// TIA Portal project "S7-1200_Conveyor_Sorting" (V17)

(* hardware
DEVICE "S7-1200 station_1"  S7-1200 Station
   slot 0: "Rack_0"  S7-1200 Rack  Rack  V1.0
   slot 1: "PLC_1"  CPU 1212C DC/DC/DC  6ES7 212-1AE40-0XB0  V4.2
DEVICE "HMI_1"  TP700 Comfort
   slot 0: "HMI_1"  TP700 Comfort  6AV2 124-0GC01-0AX0  17.0.0.0
   slot 1: "HMI_RT_1"  TP700 Comfort  6AV2 124-0GC01-0AX0  17.0.0.0
   slot 5: "HMI_1.IE_CP_1"  PROFINET Interface  17.0.0.0
      slot 1: "PROFINET Interface_1"  PROFINET Interface
         slot 1: "Port_1"  Port
         slot 2: "Port_2"  Port
   slot 7: "HMI_1.MPI/DP_CP_1"  MPI/DP Interface  17.0.0.0
*)

// ===== PLC "PLC_1"  CPU 1212C DC/DC/DC =====

VAR_GLOBAL   // PLC tag table "Default tag table"
   "StopPB" AT %I0.0 : Bool;
   "SensorEntry" AT %I0.1 : Bool;
   "SensorCheck" AT %I0.2 : Bool;
   "SensorSorter" AT %I0.3 : Bool;
   "FaultResetPB" AT %I0.4 : Bool;
   "FaultLamp" AT %Q0.0 : Bool;
   "EntryOccupiedLamp" AT %Q0.1 : Bool;
   "CheckOccupiedLamp" AT %Q0.2 : Bool;
   "SorterOccupiedLamp" AT %Q0.3 : Bool;
   "SortingActiveLamp" AT %Q0.4 : Bool;
   "Clock_Byte" AT %MB100 : Byte;
   "Clock_10Hz" AT %M100.0 : Bool;
   "Clock_5Hz" AT %M100.1 : Bool;
   "Clock_2.5Hz" AT %M100.2 : Bool;
   "Clock_2Hz" AT %M100.3 : Bool;
   "Clock_1.25Hz" AT %M100.4 : Bool;
   "Clock_1Hz" AT %M100.5 : Bool;
   "Clock_0.625Hz" AT %M100.6 : Bool;
   "Clock_0.5Hz" AT %M100.7 : Bool;
   "RemoveInvalidProduct" AT %M0.0 : Bool;
   "StartCommand" AT %M0.1 : Bool;
   "FaultResetHMI" AT %M0.2 : Bool;
END_VAR

DATA_BLOCK "Data_block_1"   // DB2
{ S7_Optimized_Access := 'TRUE' }
VERSION : 0.1
   VAR
      EntryOccupied : Bool;
      CheckOccupied : Bool;
      SorterOccupied : Bool;
      SortingActive : Bool;
      FaultActive : Bool;
      SystemRunning : Bool;
      EntryCheckTimeoutFault : Bool;
      CheckSorterTimeoutFault : Bool;
      LineStopped : Bool;
      CheckProductType : Int;
      SorterProductType : Int;
      ProductSelect : Int;
      ALine : Bool;
      BLine : Bool;
      RandomCounter : Int;
      RandomValue : Int;
      ProductACount : DInt;
      ProductBCount : DInt;
      InvalidProductFault : Bool;
      SensorCheckMemory : Bool;
      TotalProductsCount : DInt;
      AlarmWord : Word;
   END_VAR
BEGIN
END_DATA_BLOCK

// folder: System blocks/Program resources

DATA_BLOCK "IEC_Timer_0_DB_1"   // DB3
{ S7_Optimized_Access := 'TRUE' }
AUTHOR : Simatic
FAMILY : IEC
NAME : IEC_TMR
VERSION : 1.0
// stored: InstanceOfName IEC_TIMER
"IEC_TIMER"
BEGIN
END_DATA_BLOCK

DATA_BLOCK "IEC_Counter_0_DB"   // DB4
{ S7_Optimized_Access := 'TRUE' }
AUTHOR : Simatic
FAMILY : IEC
NAME : CNTR
VERSION : 1.0
// stored: InstanceOfName IEC_COUNTER
"IEC_COUNTER"
BEGIN
END_DATA_BLOCK

DATA_BLOCK "IEC_Timer_0_DB_3"   // DB5
{ S7_Optimized_Access := 'TRUE' }
AUTHOR : Simatic
FAMILY : IEC
NAME : IEC_TMR
VERSION : 1.0
// stored: InstanceOfName IEC_TIMER
"IEC_TIMER"
BEGIN
END_DATA_BLOCK

DATA_BLOCK "IEC_Timer_0_DB_4"   // DB6
{ S7_Optimized_Access := 'TRUE' }
AUTHOR : Simatic
FAMILY : IEC
NAME : IEC_TMR
VERSION : 1.0
// stored: InstanceOfName IEC_TIMER
"IEC_TIMER"
BEGIN
END_DATA_BLOCK

DATA_BLOCK "IEC_Counter_0_DB_1"   // DB7
{ S7_Optimized_Access := 'TRUE' }
AUTHOR : Simatic
FAMILY : IEC
NAME : CNTR
VERSION : 1.0
// stored: InstanceOfName IEC_COUNTER
"IEC_COUNTER"
BEGIN
END_DATA_BLOCK

DATA_BLOCK "IEC_Counter_0_DB_2"   // DB8
{ S7_Optimized_Access := 'TRUE' }
AUTHOR : Simatic
FAMILY : IEC
NAME : CNTR
VERSION : 1.0
// stored: InstanceOfName IEC_COUNTER
"IEC_COUNTER"
BEGIN
END_DATA_BLOCK

DATA_BLOCK "IEC_Timer_0_DB_2"   // DB9
{ S7_Optimized_Access := 'TRUE' }
AUTHOR : Simatic
FAMILY : IEC
NAME : IEC_TMR
VERSION : 1.0
// stored: InstanceOfName IEC_TIMER
"IEC_TIMER"
BEGIN
END_DATA_BLOCK

DATA_BLOCK "IEC_Timer_0_DB_5"   // DB10
{ S7_Optimized_Access := 'TRUE' }
AUTHOR : Simatic
FAMILY : IEC
NAME : IEC_TMR
VERSION : 1.0
// stored: InstanceOfName IEC_TIMER
"IEC_TIMER"
BEGIN
END_DATA_BLOCK

// folder: (top level)

ORGANIZATION_BLOCK "Main"   // OB1, LAD, ProgramCycle
TITLE = "Main Program Sweep (Cycle)"
{ S7_Optimized_Access := 'TRUE' }
VERSION : 0.1
   VAR_INPUT
      Initial_Call : Bool;   // Initial call of this OB
      Remanence : Bool;   // =True, if remanent data are available
   END_VAR
   VAR_TEMP   // added for the SCL form of the ladder/FBD networks
      _w1 : Bool;
      _w2 : Bool;
   END_VAR
BEGIN

REGION Network 1: Product Type Randomizer
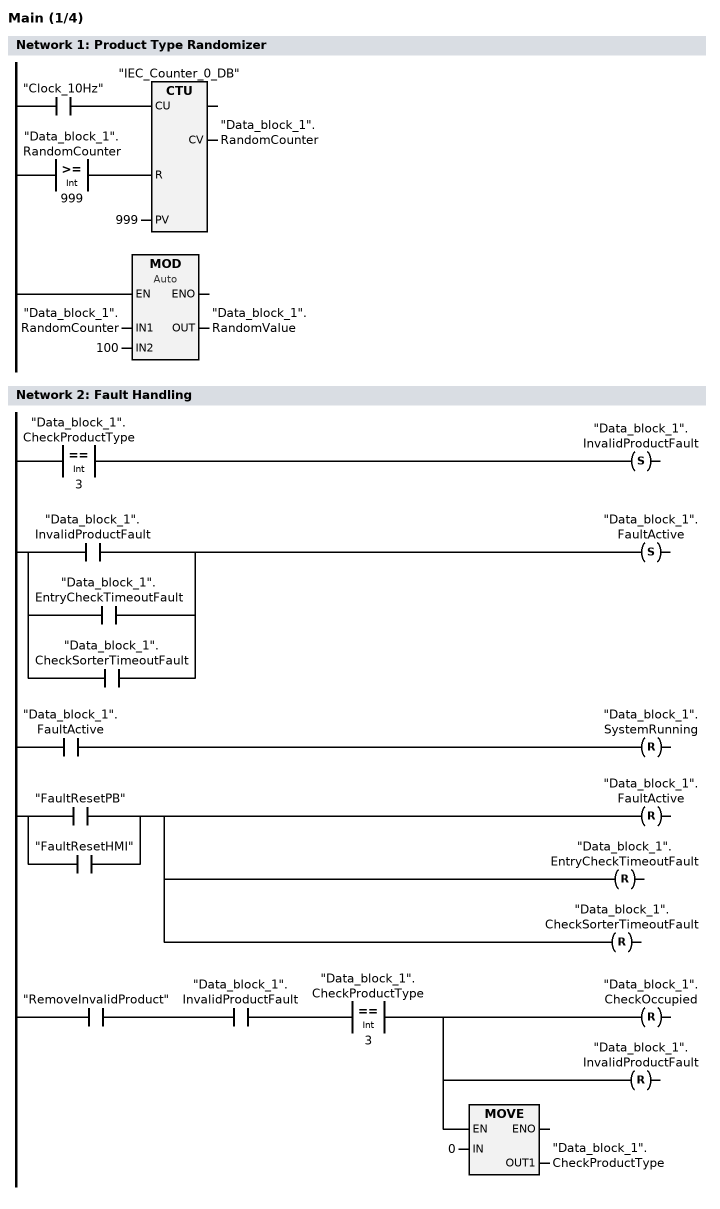
   "IEC_Counter_0_DB".CTU(CU := "Clock_10Hz",
                          R := "Data_block_1".RandomCounter >= 999,
                          PV := 999,
                          CV => "Data_block_1".RandomCounter);
   "Data_block_1".RandomValue := "Data_block_1".RandomCounter MOD 100;
END_REGION

REGION Network 2: Fault Handling
   RUNG wire#powerrail
      { S7_Templates := "SrcType := Int" } EQ_Contact(in1 := "Data_block_1".CheckProductType, in2 := 3)
      S_Coil( "Data_block_1".InvalidProductFault )
   END_RUNG
   RUNG wire#powerrail
      Contact( "Data_block_1".InvalidProductFault )
      wire#w1
      S_Coil( "Data_block_1".FaultActive )
   END_RUNG
   RUNG wire#powerrail
      Contact( "Data_block_1".EntryCheckTimeoutFault )
   END_RUNG wire#w1
   RUNG wire#powerrail
      Contact( "Data_block_1".CheckSorterTimeoutFault )
   END_RUNG wire#w1
   RUNG wire#powerrail
      Contact( "Data_block_1".FaultActive )
      R_Coil( "Data_block_1".SystemRunning )
   END_RUNG
   RUNG wire#powerrail
      Contact( "FaultResetPB" )
      wire#w2
      R_Coil( "Data_block_1".FaultActive )
   END_RUNG
   RUNG wire#powerrail
      Contact( "FaultResetHMI" )
   END_RUNG wire#w2
   RUNG wire#w2
      R_Coil( "Data_block_1".EntryCheckTimeoutFault )
   END_RUNG
   RUNG wire#w2
      R_Coil( "Data_block_1".CheckSorterTimeoutFault )
   END_RUNG
   RUNG wire#powerrail
      Contact( "RemoveInvalidProduct" )
      Contact( "Data_block_1".InvalidProductFault )
      { S7_Templates := "SrcType := Int" } EQ_Contact(in1 := "Data_block_1".CheckProductType, in2 := 3)
      wire#w3
      R_Coil( "Data_block_1".CheckOccupied )
   END_RUNG
   RUNG wire#w3
      R_Coil( "Data_block_1".InvalidProductFault )
   END_RUNG
   RUNG wire#w3
      Move(in := 0, out1 => "Data_block_1".CheckProductType)
   END_RUNG
   // the same network as SCL:
   IF "Data_block_1".CheckProductType = 3 THEN "Data_block_1".InvalidProductFault := TRUE; END_IF;
   IF "Data_block_1".InvalidProductFault OR "Data_block_1".EntryCheckTimeoutFault OR "Data_block_1".CheckSorterTimeoutFault THEN
       "Data_block_1".FaultActive := TRUE;
   END_IF;
   IF "Data_block_1".FaultActive THEN "Data_block_1".SystemRunning := FALSE; END_IF;
   IF "FaultResetPB" OR "FaultResetHMI" THEN
       "Data_block_1".FaultActive := FALSE;
       "Data_block_1".EntryCheckTimeoutFault := FALSE;
       "Data_block_1".CheckSorterTimeoutFault := FALSE;
   END_IF;
   IF "RemoveInvalidProduct" AND "Data_block_1".InvalidProductFault AND ("Data_block_1".CheckProductType = 3) THEN
       "Data_block_1".CheckOccupied := FALSE;
   END_IF;
   #_w1 := "RemoveInvalidProduct" AND "Data_block_1".InvalidProductFault AND ("Data_block_1".CheckProductType = 3);
   IF #_w1 THEN
       "Data_block_1".InvalidProductFault := FALSE;
       "Data_block_1".CheckProductType := 0;
   END_IF;
END_REGION

REGION Network 3: Alarm Word Mapping
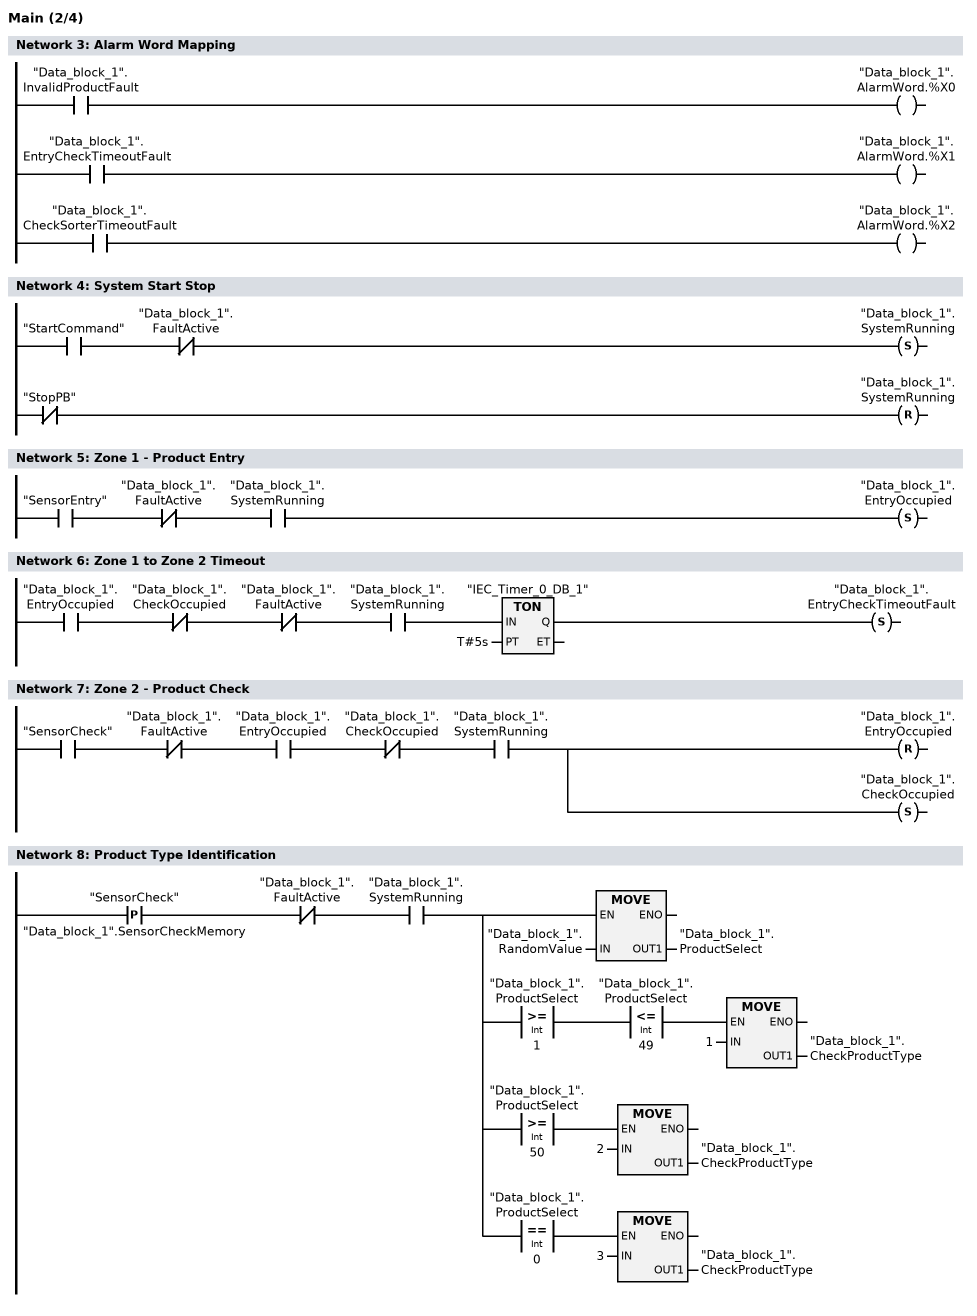
   RUNG wire#powerrail
      Contact( "Data_block_1".InvalidProductFault )
      Coil( "Data_block_1".AlarmWord.%X0 )
   END_RUNG
   RUNG wire#powerrail
      Contact( "Data_block_1".EntryCheckTimeoutFault )
      Coil( "Data_block_1".AlarmWord.%X1 )
   END_RUNG
   RUNG wire#powerrail
      Contact( "Data_block_1".CheckSorterTimeoutFault )
      Coil( "Data_block_1".AlarmWord.%X2 )
   END_RUNG
   // the same network as SCL:
   "Data_block_1".AlarmWord.%X0 := "Data_block_1".InvalidProductFault;
   "Data_block_1".AlarmWord.%X1 := "Data_block_1".EntryCheckTimeoutFault;
   "Data_block_1".AlarmWord.%X2 := "Data_block_1".CheckSorterTimeoutFault;
END_REGION

REGION Network 4: System Start Stop
   RUNG wire#powerrail
      Contact( "StartCommand" )
      I_Contact( "Data_block_1".FaultActive )
      S_Coil( "Data_block_1".SystemRunning )
   END_RUNG
   RUNG wire#powerrail
      I_Contact( "StopPB" )
      R_Coil( "Data_block_1".SystemRunning )
   END_RUNG
   // the same network as SCL:
   IF "StartCommand" AND NOT "Data_block_1".FaultActive THEN "Data_block_1".SystemRunning := TRUE; END_IF;
   IF NOT "StopPB" THEN "Data_block_1".SystemRunning := FALSE; END_IF;
END_REGION

REGION Network 5: Zone 1 - Product Entry
   RUNG wire#powerrail
      Contact( "SensorEntry" )
      I_Contact( "Data_block_1".FaultActive )
      Contact( "Data_block_1".SystemRunning )
      S_Coil( "Data_block_1".EntryOccupied )
   END_RUNG
   // the same network as SCL:
   IF "SensorEntry" AND NOT "Data_block_1".FaultActive AND "Data_block_1".SystemRunning THEN
       "Data_block_1".EntryOccupied := TRUE;
   END_IF;
END_REGION

REGION Network 6: Zone 1 to Zone 2 Timeout
   "IEC_Timer_0_DB_1".TON(IN := "Data_block_1".EntryOccupied AND NOT "Data_block_1".CheckOccupied AND NOT "Data_block_1".FaultActive AND "Data_block_1".SystemRunning,
                          PT := T#5s);
   IF "IEC_Timer_0_DB_1".Q THEN "Data_block_1".EntryCheckTimeoutFault := TRUE; END_IF;
END_REGION

REGION Network 7: Zone 2 - Product Check
   RUNG wire#powerrail
      Contact( "SensorCheck" )
      I_Contact( "Data_block_1".FaultActive )
      Contact( "Data_block_1".EntryOccupied )
      I_Contact( "Data_block_1".CheckOccupied )
      Contact( "Data_block_1".SystemRunning )
      wire#w1
      R_Coil( "Data_block_1".EntryOccupied )
   END_RUNG
   RUNG wire#w1
      S_Coil( "Data_block_1".CheckOccupied )
   END_RUNG
   // the same network as SCL:
   #_w1 := "SensorCheck" AND NOT "Data_block_1".FaultActive AND "Data_block_1".EntryOccupied AND NOT "Data_block_1".CheckOccupied AND "Data_block_1".SystemRunning;
   IF #_w1 THEN
       "Data_block_1".EntryOccupied := FALSE;
       "Data_block_1".CheckOccupied := TRUE;
   END_IF;
END_REGION

REGION Network 8: Product Type Identification
   RUNG wire#powerrail
      P_Contact(operand := "SensorCheck", bit := "Data_block_1".SensorCheckMemory)
      I_Contact( "Data_block_1".FaultActive )
      Contact( "Data_block_1".SystemRunning )
      wire#w1
      Move(in := "Data_block_1".RandomValue, out1 => "Data_block_1".ProductSelect)
   END_RUNG
   RUNG wire#w1
      { S7_Templates := "SrcType := Int" } GE_Contact(in1 := "Data_block_1".ProductSelect, in2 := 1)
      { S7_Templates := "SrcType := Int" } LE_Contact(in1 := "Data_block_1".ProductSelect, in2 := 49)
      Move(in := 1, out1 => "Data_block_1".CheckProductType)
   END_RUNG
   RUNG wire#w1
      { S7_Templates := "SrcType := Int" } GE_Contact(in1 := "Data_block_1".ProductSelect, in2 := 50)
      Move(in := 2, out1 => "Data_block_1".CheckProductType)
   END_RUNG
   RUNG wire#w1
      { S7_Templates := "SrcType := Int" } EQ_Contact(in1 := "Data_block_1".ProductSelect, in2 := 0)
      Move(in := 3, out1 => "Data_block_1".CheckProductType)
   END_RUNG
   // the same network as SCL:
   #_w1 := "SensorCheck" AND NOT "Data_block_1".SensorCheckMemory;   // rising edge of "SensorCheck"
   "Data_block_1".SensorCheckMemory := "SensorCheck";
   #_w2 := #_w1 AND NOT "Data_block_1".FaultActive AND "Data_block_1".SystemRunning;
   IF #_w2 THEN "Data_block_1".ProductSelect := "Data_block_1".RandomValue; END_IF;
   IF #_w2 AND ("Data_block_1".ProductSelect >= 1) AND ("Data_block_1".ProductSelect <= 49) THEN
       "Data_block_1".CheckProductType := 1;
   END_IF;
   IF #_w2 AND ("Data_block_1".ProductSelect >= 50) THEN "Data_block_1".CheckProductType := 2; END_IF;
   IF #_w2 AND ("Data_block_1".ProductSelect = 0) THEN "Data_block_1".CheckProductType := 3; END_IF;
END_REGION

REGION Network 9: Zone 2 to Zone 3 Timeout
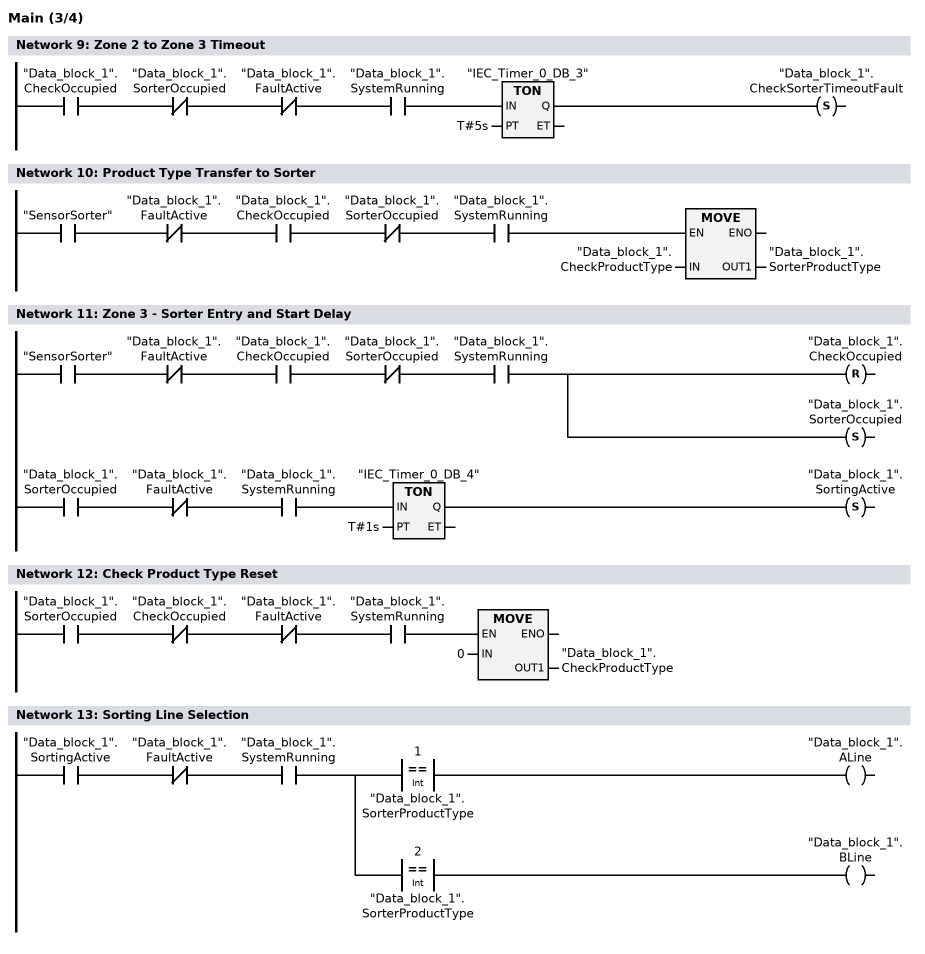
   "IEC_Timer_0_DB_3".TON(IN := "Data_block_1".CheckOccupied AND NOT "Data_block_1".SorterOccupied AND NOT "Data_block_1".FaultActive AND "Data_block_1".SystemRunning,
                          PT := T#5s);
   IF "IEC_Timer_0_DB_3".Q THEN "Data_block_1".CheckSorterTimeoutFault := TRUE; END_IF;
END_REGION

REGION Network 10: Product Type Transfer to Sorter
   RUNG wire#powerrail
      Contact( "SensorSorter" )
      I_Contact( "Data_block_1".FaultActive )
      Contact( "Data_block_1".CheckOccupied )
      I_Contact( "Data_block_1".SorterOccupied )
      Contact( "Data_block_1".SystemRunning )
      Move(in := "Data_block_1".CheckProductType, out1 => "Data_block_1".SorterProductType)
   END_RUNG
   // the same network as SCL:
   IF "SensorSorter" AND NOT "Data_block_1".FaultActive AND "Data_block_1".CheckOccupied AND NOT "Data_block_1".SorterOccupied AND "Data_block_1".SystemRunning THEN
       "Data_block_1".SorterProductType := "Data_block_1".CheckProductType;
   END_IF;
END_REGION

REGION Network 11: Zone 3 - Sorter Entry and Start Delay
   #_w1 := "SensorSorter" AND NOT "Data_block_1".FaultActive AND "Data_block_1".CheckOccupied AND NOT "Data_block_1".SorterOccupied AND "Data_block_1".SystemRunning;
   IF #_w1 THEN
       "Data_block_1".CheckOccupied := FALSE;
       "Data_block_1".SorterOccupied := TRUE;
   END_IF;
   "IEC_Timer_0_DB_4".TON(IN := "Data_block_1".SorterOccupied AND NOT "Data_block_1".FaultActive AND "Data_block_1".SystemRunning,
                          PT := T#1s);
   IF "IEC_Timer_0_DB_4".Q THEN "Data_block_1".SortingActive := TRUE; END_IF;
END_REGION

REGION Network 12: Check Product Type Reset
   RUNG wire#powerrail
      Contact( "Data_block_1".SorterOccupied )
      I_Contact( "Data_block_1".CheckOccupied )
      I_Contact( "Data_block_1".FaultActive )
      Contact( "Data_block_1".SystemRunning )
      Move(in := 0, out1 => "Data_block_1".CheckProductType)
   END_RUNG
   // the same network as SCL:
   IF "Data_block_1".SorterOccupied AND NOT "Data_block_1".CheckOccupied AND NOT "Data_block_1".FaultActive AND "Data_block_1".SystemRunning THEN
       "Data_block_1".CheckProductType := 0;
   END_IF;
END_REGION

REGION Network 13: Sorting Line Selection
   RUNG wire#powerrail
      Contact( "Data_block_1".SortingActive )
      I_Contact( "Data_block_1".FaultActive )
      Contact( "Data_block_1".SystemRunning )
      wire#w1
      { S7_Templates := "SrcType := Int" } EQ_Contact(in1 := 1, in2 := "Data_block_1".SorterProductType)
      Coil( "Data_block_1".ALine )
   END_RUNG
   RUNG wire#w1
      { S7_Templates := "SrcType := Int" } EQ_Contact(in1 := 2, in2 := "Data_block_1".SorterProductType)
      Coil( "Data_block_1".BLine )
   END_RUNG
   // the same network as SCL:
   #_w1 := "Data_block_1".SortingActive AND NOT "Data_block_1".FaultActive AND "Data_block_1".SystemRunning;
   "Data_block_1".ALine := #_w1 AND (1 = "Data_block_1".SorterProductType);
   "Data_block_1".BLine := #_w1 AND (2 = "Data_block_1".SorterProductType);
END_REGION

REGION Network 14: Sorting Process and Counters
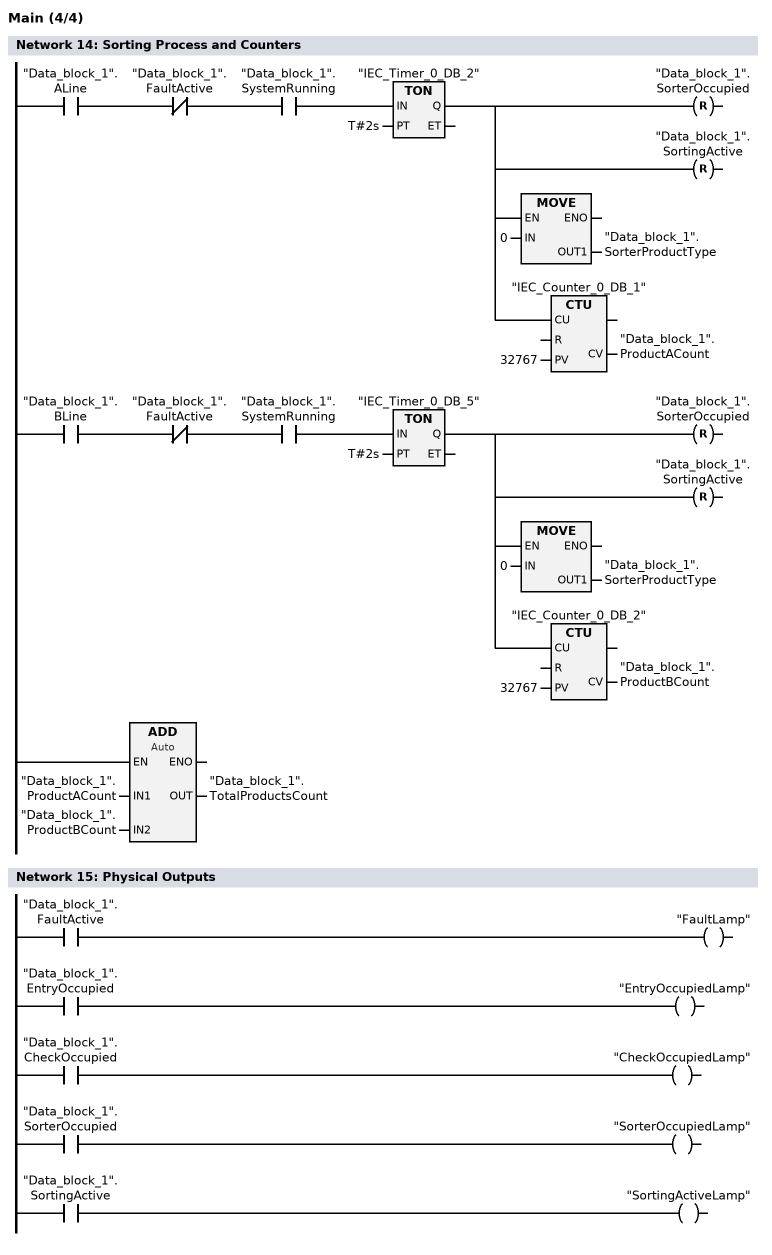
   "IEC_Timer_0_DB_2".TON(IN := "Data_block_1".ALine AND NOT "Data_block_1".FaultActive AND "Data_block_1".SystemRunning,
                          PT := T#2s);
   IF "IEC_Timer_0_DB_2".Q THEN
       "Data_block_1".SorterOccupied := FALSE;
       "Data_block_1".SortingActive := FALSE;
       "Data_block_1".SorterProductType := 0;
   END_IF;
   "IEC_Counter_0_DB_1".CTU(CU := "IEC_Timer_0_DB_2".Q, PV := 32767, CV => "Data_block_1".ProductACount);
   "IEC_Timer_0_DB_5".TON(IN := "Data_block_1".BLine AND NOT "Data_block_1".FaultActive AND "Data_block_1".SystemRunning,
                          PT := T#2s);
   IF "IEC_Timer_0_DB_5".Q THEN
       "Data_block_1".SorterOccupied := FALSE;
       "Data_block_1".SortingActive := FALSE;
       "Data_block_1".SorterProductType := 0;
   END_IF;
   "IEC_Counter_0_DB_2".CTU(CU := "IEC_Timer_0_DB_5".Q, PV := 32767, CV => "Data_block_1".ProductBCount);
   "Data_block_1".TotalProductsCount := "Data_block_1".ProductACount + "Data_block_1".ProductBCount;
END_REGION

REGION Network 15: Physical Outputs
   RUNG wire#powerrail
      Contact( "Data_block_1".FaultActive )
      Coil( "FaultLamp" )
   END_RUNG
   RUNG wire#powerrail
      Contact( "Data_block_1".EntryOccupied )
      Coil( "EntryOccupiedLamp" )
   END_RUNG
   RUNG wire#powerrail
      Contact( "Data_block_1".CheckOccupied )
      Coil( "CheckOccupiedLamp" )
   END_RUNG
   RUNG wire#powerrail
      Contact( "Data_block_1".SorterOccupied )
      Coil( "SorterOccupiedLamp" )
   END_RUNG
   RUNG wire#powerrail
      Contact( "Data_block_1".SortingActive )
      Coil( "SortingActiveLamp" )
   END_RUNG
   // the same network as SCL:
   "FaultLamp" := "Data_block_1".FaultActive;
   "EntryOccupiedLamp" := "Data_block_1".EntryOccupied;
   "CheckOccupiedLamp" := "Data_block_1".CheckOccupied;
   "SorterOccupiedLamp" := "Data_block_1".SorterOccupied;
   "SortingActiveLamp" := "Data_block_1".SortingActive;
END_REGION
END_ORGANIZATION_BLOCK

(* ===== HMI "HMI_RT_1" =====
system functions are stored by id; their names below are inferred from use
connection "HMI_Connection_2": ETHERNET, S7_1200_OMS

HMI tags "Default tag table"
   "Data_block_1_SystemRunning" : Bool = PLC Data_block_1.SystemRunning, 1 s
   "Data_block_1_FaultActive" : Bool = PLC Data_block_1.FaultActive, 1 s
   "CheckOccupiedLamp" : Bool = PLC CheckOccupiedLamp AT %Q0.2, 1 s
   "EntryOccupiedLamp" : Bool = PLC EntryOccupiedLamp AT %Q0.1, 1 s
   "SorterOccupiedLamp" : Bool = PLC SorterOccupiedLamp AT %Q0.3, 1 s
   "Data_block_1_CheckProductType" : Int = PLC Data_block_1.CheckProductType, 1 s
   "Data_block_1_SorterProductType" : Int = PLC Data_block_1.SorterProductType, 1 s
   "RemoveInvalidProduct" : Bool = PLC RemoveInvalidProduct AT %M0.0, 1 s
   "Data_block_1_ALine" : Bool = PLC Data_block_1.ALine, 1 s
   "Data_block_1_BLine" : Bool = PLC Data_block_1.BLine, 1 s
   "SensorCheck" : Bool = PLC SensorCheck AT %I0.2, 1 s
   "SensorSorter" : Bool = PLC SensorSorter AT %I0.3, 1 s
   "Data_block_1_TotalProductsCount" : DInt = PLC Data_block_1.TotalProductsCount, 1 s
   "Data_block_1_ProductACount" : DInt = PLC Data_block_1.ProductACount, 1 s
   "Data_block_1_ProductBCount" : DInt = PLC Data_block_1.ProductBCount, 1 s
   "Data_block_1_InvalidProductFault" : Bool = PLC Data_block_1.InvalidProductFault AT %DB1.DBX0.0, 1 s
   "Data_block_1_AlarmWord" : Word = PLC Data_block_1.AlarmWord, 1 s
   "FaultResetPB" : Bool = PLC FaultResetPB AT %I0.4, 1 s
   "FaultResetHMI" : Bool = PLC FaultResetHMI AT %M0.2, 1 s
   "StopPB" : Bool = PLC StopPB AT %I0.0, 1 s
   "SensorEntry" : Bool = PLC SensorEntry AT %I0.1, 1 s
   "FaultLamp" : Bool = PLC FaultLamp AT %Q0.0, 1 s
   "SortingActiveLamp" : Bool = PLC SortingActiveLamp AT %Q0.4, 1 s
   "Data_block_1_EntryOccupied" : Bool = PLC Data_block_1.EntryOccupied, 1 s
   "Data_block_1_CheckOccupied" : Bool = PLC Data_block_1.CheckOccupied, 1 s
   "Data_block_1_SorterOccupied" : Bool = PLC Data_block_1.SorterOccupied, 1 s
   "Data_block_1_SortingActive" : Bool = PLC Data_block_1.SortingActive, 1 s
   "Data_block_1_Zone1-Zone2Fault" : Bool = PLC Data_block_1.EntryCheckTimeoutFault, 1 s
   "Data_block_1_Zone2-Zone3Fault" : Bool = PLC Data_block_1.CheckSorterTimeoutFault, 1 s
   "StartCommand" : Bool = PLC StartCommand AT %M0.1, 1 s

discrete alarms
   1: 'Invalid product detected - remove product and reset fault', class Errors, trigger "Data_block_1_AlarmWord" bit 0
   2: 'Product timeout between ENTRY and CHECK', class Errors, trigger "Data_block_1_AlarmWord" bit 1
   3: 'Product timeout between CHECK and SORTER', class Errors, trigger "Data_block_1_AlarmWord" bit 2

graphic list "@DiagnosticsStates": 0 '@Diagnostics_StateGood'; 1 '@Diagnostics_StateBad'

Template "Template_1" 800x480
   Button "Exit" at 720,420 size 78x58; TextOff 'Exit'; PictureOff "ExitRuntime_TP700_Comfort_TR"; PictureOn "ExitRuntime_TP700_Comfort_TR"
      on Release: StopRuntime(0)
   Button "Template_Button_6" at 161,420 size 126x58; TextOff 'DIAGNOSTICS'
      on Click: ActivateScreen("Diagnostics", 0)
   Button "Template_Button_7" at 81,420 size 78x58; TextOff 'ALARMS'
      on Click: ActivateScreen("Alarms", 0)
   Button "Start screen" at 1,420 size 78x58; TextOff 'Start screen'; PictureOff "NavigateHome_TP700_Comfort_TR"; PictureOn "NavigateHome_TP700_Comfort_TR"
      on Click: ActivateScreen("Root screen", 0)

screen "Root screen" 800x480, template "Template_1"
   TextField "HmiScreenItemData" at 6,108 size 640x25; Text 'Text'
   TextField "Text field_1" at 218,1 size 402x34; Text 'CONVEYOR SORTING SYSTEM'
   TextField "Text field_2" at 13,40 size 84x23; Text 'SYSTEM:'
   TextField "Text field_3" at 90,40 size 89x23; Text 'STOPPED'
      Visibility <- "Data_block_1_SystemRunning"
      Appearance <- "Data_block_1_SystemRunning"
   TextField "Text field_4" at 90,40 size 91x23; Text 'RUNNING'
      Visibility <- "Data_block_1_SystemRunning"
      Appearance <- "Data_block_1_SystemRunning"
   Button "Button_1" at 47,76 size 96x32; TextOff 'START'
      on Press: SetBit("StartCommand")
      Visibility <- "Data_block_1_FaultActive"
      on Release: ResetBit("StartCommand")
   Button "Button_2" at 47,117 size 96x32; TextOff 'STOP'
      on Press: ResetBit("Data_block_1_SystemRunning")
      Visibility <- "Data_block_1_FaultActive"
   TextField "Text field_5" at 542,40 size 70x23; Text 'FAULT:'
   TextField "Text field_6" at 612,40 size 31x23; Text 'NO'
      Appearance <- "Data_block_1_FaultActive"
      Visibility <- "Data_block_1_FaultActive"
   TextField "Text field_7" at 604,40 size 73x23; Text 'ACTIVE'
      Appearance <- "Data_block_1_FaultActive"
      Visibility <- "Data_block_1_FaultActive"
   Circle "Circle_1" at 671,28 size 48x48
      Appearance <- "Data_block_1_FaultActive"
      Visibility <- "Data_block_1_FaultActive"
   Polygon "Polygon_2" at 572,298 size 21x14
      Appearance <- "Data_block_1_BLine"
   Polygon "Polygon_3" at 477,298 size 21x14
      Appearance <- "Data_block_1_ALine"
   TextField "Text field_8" at 555,312 size 65x23; Text 'B LINE'
   TextField "Text field_9" at 462,312 size 66x23; Text 'A LINE'
   Polygon "Polygon_4" at 320,199 size 13x20
      Appearance <- "SensorCheck"
   Polygon "Polygon_5" at 474,199 size 13x20
      Appearance <- "SensorSorter"
   TextField "Text field_10" at 186,199 size 93x23; Text 'PRODUCT'
   TextField "Text field_11" at 339,199 size 93x23; Text 'PRODUCT'
   TextField "Text field_12" at 492,199 size 93x23; Text 'PRODUCT'
   Circle "Circle_2" at 213,149 size 30x30
      Appearance <- "EntryOccupiedLamp"
   Circle "Circle_3" at 367,149 size 30x30
      Appearance <- "CheckOccupiedLamp"
   Circle "Circle_4" at 521,149 size 30x30
      Appearance <- "SorterOccupiedLamp"
   TextField "Text field_13" at 197,117 size 66x23; Text 'ENTRY'
   TextField "Text field_14" at 352,117 size 65x23; Text 'CHECK'
   TextField "Text field_15" at 498,117 size 78x23; Text 'SORTER'
   TextField "Text field_16" at 373,151 size 18x23; Text 'A'
      Visibility <- "Data_block_1_CheckProductType"
   TextField "Text field_17" at 528,151 size 18x23; Text 'A'
      Visibility <- "Data_block_1_SorterProductType"
   TextField "Text field_18" at 374,151 size 17x23; Text 'B'
      Visibility <- "Data_block_1_CheckProductType"
   TextField "Text field_19" at 529,151 size 17x23; Text 'B'
      Visibility <- "Data_block_1_SorterProductType"
   TextField "Text field_20" at 373,151 size 17x23; Text 'C'
      Visibility <- "Data_block_1_CheckProductType"
   TextField "Text field_21" at 29,280 size 78x23; Text 'TOTAL:'
   TextField "Text field_22" at 29,332 size 125x23; Text 'PRODUCT A:'
   TextField "Text field_23" at 29,374 size 124x23; Text 'PRODUCT B:'
   IOField "I/O field_1" at 97,276 size 96x32; FormatPattern 999999
      ProcessValue <- "Data_block_1_TotalProductsCount"
   IOField "I/O field_2" at 143,327 size 96x32; FormatPattern 999999
      ProcessValue <- "Data_block_1_ProductACount"
   IOField "I/O field_3" at 143,369 size 96x32; FormatPattern 999999
      ProcessValue <- "Data_block_1_ProductBCount"

screen "Alarms" 800x480, template "Template_1"
   TextField "Text field_1" at 260,9 size 266x23; Text 'ALARMS & FAULT HANDLING'
   AlarmView "Alarm view_1" at 23,98 size 761x241
   TextField "Text field_5" at 523,49 size 70x23; Text 'FAULT:'
   TextField "Text field_6" at 593,49 size 31x23; Text 'NO'
      Visibility <- "Data_block_1_FaultActive"
      Appearance <- "Data_block_1_FaultActive"
   TextField "Text field_7" at 585,49 size 73x23; Text 'ACTIVE'
      Visibility <- "Data_block_1_FaultActive"
      Appearance <- "Data_block_1_FaultActive"
   Circle "Circle_1" at 652,37 size 48x48
      Visibility <- "Data_block_1_FaultActive"
      Appearance <- "Data_block_1_FaultActive"
   TextField "Text field_2" at 98,49 size 84x23; Text 'SYSTEM:'
   TextField "Text field_3" at 175,49 size 89x23; Text 'STOPPED'
      Visibility <- "Data_block_1_SystemRunning"
      Appearance <- "Data_block_1_SystemRunning"
   TextField "Text field_4" at 175,49 size 91x23; Text 'RUNNING'
      Visibility <- "Data_block_1_SystemRunning"
      Appearance <- "Data_block_1_SystemRunning"
   Button "Button_1" at 151,379 size 96x32; TextOff 'RESET'
      on Press: SetBit("FaultResetHMI")
      on Release: ResetBit("FaultResetHMI")
      Visibility <- "Data_block_1_FaultActive"
   Button "Button_2" at 497,379 size 96x32; TextOff 'REMOVE'
      on Press: SetBit("RemoveInvalidProduct")
      on Release: ResetBit("RemoveInvalidProduct")
      Visibility <- "Data_block_1_InvalidProductFault"
   TextField "Text field_8" at 140,356 size 127x23; Text 'FAULT RESET'
      Visibility <- "Data_block_1_FaultActive"
   TextField "Text field_9" at 434,356 size 257x23; Text 'REMOVE INVALID PRODUCT'
      Visibility <- "Data_block_1_InvalidProductFault"

screen "Diagnostics" 800x480, template "Template_1"
   TextField "Text field_1" at 334,13 size 132x23; Text 'DIAGNOSTICS'
   TextField "Text field_2" at 40,51 size 157x23; Text 'DIGITAL INPUTS'
   TextField "Text field_3" at 38,84 size 76x23; Text 'Stop PB'
   TextField "Text field_4" at 38,111 size 120x23; Text 'Entry Sensor'
   TextField "Text field_5" at 38,138 size 126x23; Text 'Check Sensor'
   TextField "Text field_6" at 40,165 size 129x23; Text 'Sorter Sensor'
   TextField "Text field_7" at 40,191 size 109x23; Text 'Fault Reset'
   Circle "Circle_1" at 109,83 size 26x26
      Appearance <- "StopPB"
   Circle "Circle_2" at 147,108 size 26x26
      Appearance <- "SensorEntry"
   Circle "Circle_3" at 153,136 size 26x26
      Appearance <- "SensorCheck"
   Circle "Circle_4" at 157,164 size 26x26
      Appearance <- "SensorSorter"
   Circle "Circle_5" at 139,188 size 26x26
      Appearance <- "FaultResetPB"
   TextField "Text field_8" at 270,49 size 174x23; Text 'DIGITAL OUTPUTS'
   TextField "Text field_9" at 270,97 size 178x23; Text 'Entry Stage Yellow'
   TextField "Text field_10" at 270,120 size 177x23; Text 'Check Stage Green'
   TextField "Text field_11" at 270,143 size 179x23; Text 'Sorter Stage White'
   TextField "Text field_12" at 270,74 size 105x23; Text 'Fault Lamp'
   TextField "Text field_13" at 270,166 size 125x23; Text 'Sorting Lamp'
   Circle "Circle_6" at 365,72 size 26x26
      Appearance <- "FaultLamp"
   Circle "Circle_7" at 430,92 size 26x26
      Appearance <- "EntryOccupiedLamp"
   Circle "Circle_8" at 430,118 size 26x26
      Appearance <- "CheckOccupiedLamp"
   Circle "Circle_9" at 430,144 size 26x26
      Appearance <- "SorterOccupiedLamp"
   Circle "Circle_10" at 389,164 size 26x26
      Appearance <- "SortingActiveLamp"
   TextField "Text field_15" at 519,49 size 166x23; Text 'PROCESS STATUS'
   TextField "Text field_16" at 517,118 size 140x23; Text 'Entry Occupied'
   TextField "Text field_17" at 517,143 size 146x23; Text 'Check Occupied'
   TextField "Text field_18" at 517,166 size 149x23; Text 'Sorter Occupied'
   TextField "Text field_19" at 519,233 size 185x23; Text 'Check Product Type'
   TextField "Text field_20" at 519,271 size 188x23; Text 'Sorter Product Type'
   TextField "Text field_21" at 517,190 size 134x23; Text 'Sorting Active'
   TextField "Text field_22" at 519,76 size 150x23; Text 'System Running'
   TextField "Text field_23" at 270,257 size 114x23; Text 'Fault Active'
   Circle "Circle_12" at 656,76 size 26x26
      Appearance <- "Data_block_1_SystemRunning"
   Circle "Circle_13" at 645,114 size 26x26
      Appearance <- "Data_block_1_EntryOccupied"
   Circle "Circle_14" at 648,140 size 26x26
      Appearance <- "Data_block_1_CheckOccupied"
   Circle "Circle_15" at 649,166 size 26x26
      Appearance <- "Data_block_1_SorterOccupied"
   Circle "Circle_16" at 636,189 size 26x26
      Appearance <- "Data_block_1_SortingActive"
   Circle "Circle_17" at 371,253 size 26x26
      Appearance <- "Data_block_1_FaultActive"
   TextField "Text field_24" at 699,233 size 18x23; Text 'A'
      Visibility <- "Data_block_1_CheckProductType"
   TextField "Text field_25" at 700,233 size 17x23; Text 'B'
      Visibility <- "Data_block_1_CheckProductType"
   TextField "Text field_26" at 699,233 size 17x23; Text 'C'
      Visibility <- "Data_block_1_CheckProductType"
   TextField "Text field_27" at 698,271 size 18x23; Text 'A'
      Visibility <- "Data_block_1_SorterProductType"
   TextField "Text field_28" at 699,271 size 17x23; Text 'B'
      Visibility <- "Data_block_1_SorterProductType"
   TextField "Text field_29" at 40,262 size 78x23; Text 'TOTAL:'
   TextField "Text field_30" at 40,314 size 125x23; Text 'PRODUCT A:'
   TextField "Text field_31" at 40,356 size 124x23; Text 'PRODUCT B:'
   IOField "I/O field_1" at 108,258 size 96x32; FormatPattern 999999
      ProcessValue <- "Data_block_1_TotalProductsCount"
   IOField "I/O field_2" at 154,309 size 96x32; FormatPattern 999999
      ProcessValue <- "Data_block_1_ProductACount"
   IOField "I/O field_3" at 154,351 size 96x32; FormatPattern 999999
      ProcessValue <- "Data_block_1_ProductBCount"
   TextField "Text field_14" at 270,233 size 74x23; Text 'FAULTS'
   TextField "Text field_32" at 270,285 size 144x23; Text 'Invalid Product'
   TextField "Text field_33" at 270,316 size 196x23; Text 'Entry-Check Timeout'
   TextField "Text field_34" at 269,346 size 205x23; Text 'Check-Sorter Timeout'
   Circle "Circle_11" at 400,282 size 26x26
      Appearance <- "Data_block_1_InvalidProductFault"
   Circle "Circle_20" at 448,314 size 26x26
      Appearance <- "Data_block_1_Zone1-Zone2Fault"
   Circle "Circle_21" at 453,342 size 26x26
      Appearance <- "Data_block_1_Zone2-Zone3Fault"
   TextField "Text field_35" at 40,234 size 103x23; Text 'COUNTERS'
*)